PROGRAM MAIN
VAR
END_VAR

END_PROGRAM

(* stored: Version 1.1.0.1
   POU MAIN: Id {af0b725c-f20d-4cbb-ae2a-d59e7a1d6f81} *)
